(* PLC project servo_velocity, Dassault Systèmes ControlBuild 2024x *)
(* stored: creationDateTime 2023-10-04T11:03:54-01:00 *)

(* This module controls velocity behavior of the motion drive *)
FUNCTION_BLOCK motion_control.servo_velocity
  VAR_INPUT
    MoveVelEnable : BOOL := false;
    MoveVelStart : BOOL := false;
    MoveSpeed : REAL := 100.0;
    MoveAcceleration : REAL := 100.0;
    MoveDeceleration : REAL := 100.0;
    MAX_SPEED : REAL(0.0..3.4e+38) := 1000.0;
    MAX_ACCEL : REAL(0.0..3.4e+38) := 300.0;
    MAX_DECEL : REAL(0.0..3.4e+38) := 300.0;
    MODULO_LENGTH : REAL := 0.0;
  END_VAR
  VAR_IN_OUT
    status : INT := 0;
    errorFlag : INT := 0;
    MoveVelDone : BOOL := false;
    ActualPositionAx : REAL := 0.0;
    ActualVelocity : REAL := 0.0;
  END_VAR
  VAR
    firstStep : BOOL := true;
    stepDone : BOOL := false;
    currentTime : REAL := 0.0;
    MoveSpeed1 : REAL := 0.0;
    acceleration : REAL := 0.0;
    deceleration : REAL := 0.0;
    orderSpeed : REAL := 0.0;
    endChangeSpeed : REAL := 0.0;
    accelDecelChangeSpeed : REAL := 0.0;
    ActualVelocity1 : REAL := 0.0;
    speedChanged : BOOL := false;
  END_VAR


ACTION C_source_code:
/* ----------------------------------------------------------------	*/
/* Type : Model of Operative Behaviour					*/
/* Category :  motion control						*/
/* Author : 									*/
/* Update date : June 2021							*/
/* ----------------------------------------------------------------	*/
/* This module controls velocity behavior of the motion drive	 	*/
/* ----------------------------------------------------------------	*/

stepDone = 0;
if (MoveVelEnable) {
	if (status == 0) {
		stepDone = 1;
		if (MoveVelStart == 1) {
			errorFlag = 0;
			if (!(MoveAcceleration > 0 && MoveAcceleration <= 100.0)) {
				errorFlag = 1;
			}
			if (!(MoveDeceleration > 0 && MoveDeceleration <= 100.0)) {
				errorFlag = 2;
			}
			if (!(MoveSpeed >= -100.0 && MoveSpeed <= 100.0)) {
				errorFlag = 3;
			}
			if (errorFlag == 0) {
				status = 1;
				MoveVelDone = 0;
				ActualVelocity = 0;
				speedChanged = 1;
			}
		}
	}
	if (status != 0) {
		if (MoveSpeed1 != MoveSpeed || speedChanged != 0) {
			speedChanged = 0;
			currentTime = 0;
			orderSpeed = MoveSpeed * MAX_SPEED / 100.0;
			if (MoveSpeed >= 0) {
				acceleration = +MoveAcceleration * MAX_ACCEL / 100.0;
				deceleration = +MoveDeceleration * -MAX_DECEL / 100.0;
				accelDecelChangeSpeed = ActualVelocity > orderSpeed  ? deceleration : acceleration;
			} else {
				acceleration = -MoveAcceleration * MAX_ACCEL / 100.0; 
				deceleration = -MoveDeceleration * -MAX_DECEL / 100.0;
				accelDecelChangeSpeed = ActualVelocity > orderSpeed  ? acceleration : deceleration;
			}
			endChangeSpeed = fabs((orderSpeed - ActualVelocity) / accelDecelChangeSpeed);
			status = 1;
		}
	}
	if (status == 1 && stepDone == 0) { // CHANGE SPEED
		stepDone = 1;
		ActualVelocity = ActualVelocity + accelDecelChangeSpeed * CLOCK_PERIOD/1000000;
		if (currentTime > endChangeSpeed) {
			ActualVelocity = orderSpeed;
			status = 2;
		}
		if (MoveVelStart == 0) {
			status = 3;
		}
	}
	if (status == 2 && stepDone == 0) { // CONSTANT SPEED
		stepDone = 1;
		ActualVelocity = orderSpeed;
		if (MoveVelStart == 0) {
			status = 3;
		}
	}
	if (status == 3 && stepDone == 0) { // DECELERATION TO STOP
		stepDone = 1;
		ActualVelocity = ActualVelocity + deceleration * CLOCK_PERIOD/1000000;
		if (ActualVelocity1 * ActualVelocity <= 0.0) {
			ActualVelocity = 0.0;
			status = 4;
		}
		if (MoveVelStart != 0) {
			status = 1;
			speedChanged = 1;
		}
	}
	if (status == 4 && stepDone == 0) { // END
		stepDone = 1;
		ActualVelocity = 0.0;
		status = 0;
		MoveVelDone = 1;
	}
	if (status != 0) {
		ActualPositionAx = ActualPositionAx + ActualVelocity * CLOCK_PERIOD/1000000;
		if (MODULO_LENGTH != 0.0 ) {
			if (ActualPositionAx > MODULO_LENGTH) {
				ActualPositionAx = ActualPositionAx - MODULO_LENGTH;
			}
			if (ActualPositionAx < 0.0) {
				ActualPositionAx = ActualPositionAx + MODULO_LENGTH;
			}
			if (fabs(ActualVelocity * CLOCK_PERIOD/1000000) > MODULO_LENGTH/2.0) {
				errorFlag = 4;
			}
		}
	}
}

ActualVelocity1 = ActualVelocity;
MoveSpeed1 = MoveSpeed;
currentTime += CLOCK_PERIOD/1000000;

firstStep = 0;
END_ACTION
END_FUNCTION_BLOCK
